// SIMATIC S7-200 project (STEP 7-Micro/WIN), CPU 221 REL 01.10

ORGANIZATION_BLOCK MAIN:OB1
TITLE=PROGRAM COMMENTS
BEGIN
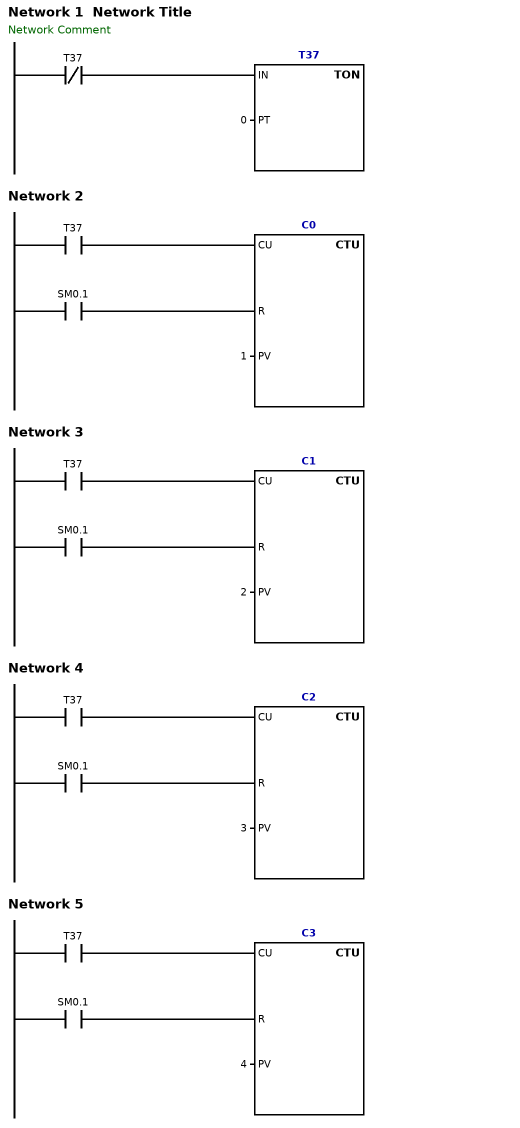
Network 1 // Network Title
// Network Comment
// (network saved uncompiled; LAD cells follow)
// row 0: c0 -|/|- T37  c1 --  c2 [TON T37 IN:=power@row0, PT:=0]
// row 1: c2 [box]
Network 2
LD     T37
LD     SM0.1
CTU    C0, 1
Network 3
LD     T37
LD     SM0.1
CTU    C1, 2
Network 4
LD     T37
LD     SM0.1
CTU    C2, 3
Network 5
LD     T37
LD     SM0.1
CTU    C3, 4
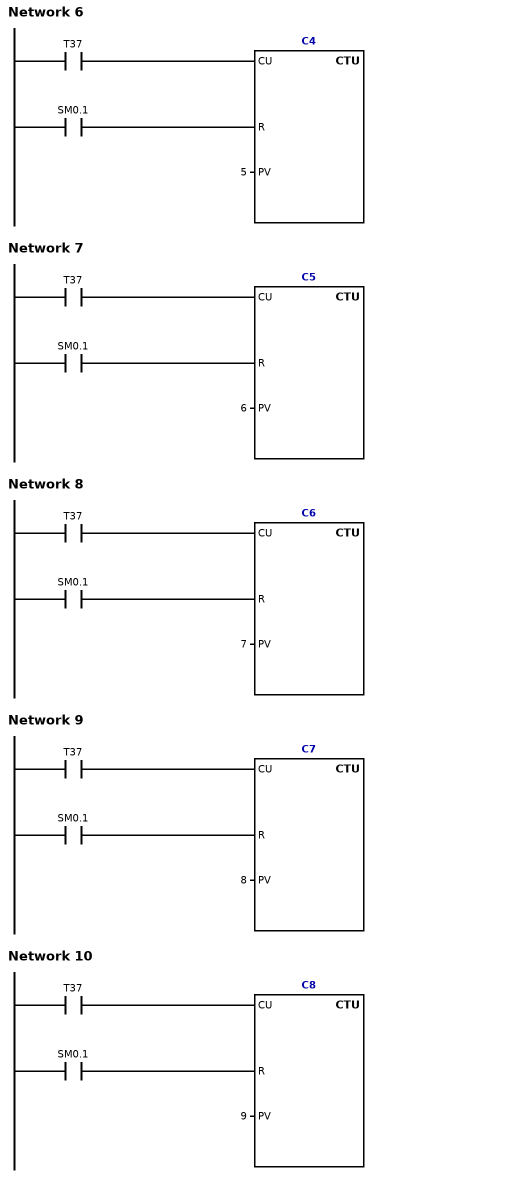
Network 6
LD     T37
LD     SM0.1
CTU    C4, 5
Network 7
LD     T37
LD     SM0.1
CTU    C5, 6
Network 8
LD     T37
LD     SM0.1
CTU    C6, 7
Network 9
LD     T37
LD     SM0.1
CTU    C7, 8
Network 10
LD     T37
LD     SM0.1
CTU    C8, 9
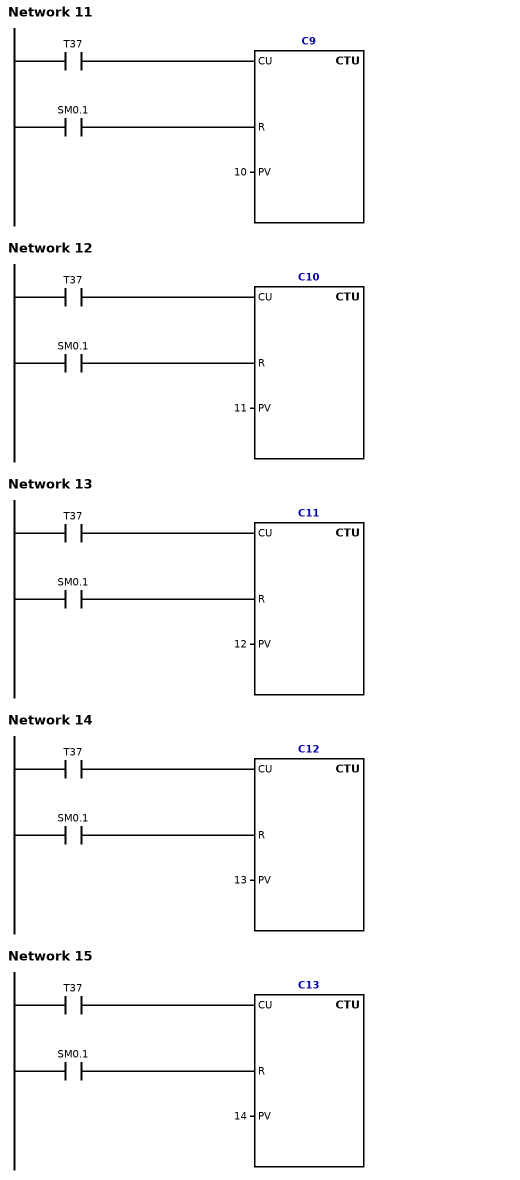
Network 11
LD     T37
LD     SM0.1
CTU    C9, 10
Network 12
LD     T37
LD     SM0.1
CTU    C10, 11
Network 13
LD     T37
LD     SM0.1
CTU    C11, 12
Network 14
LD     T37
LD     SM0.1
CTU    C12, 13
Network 15
LD     T37
LD     SM0.1
CTU    C13, 14
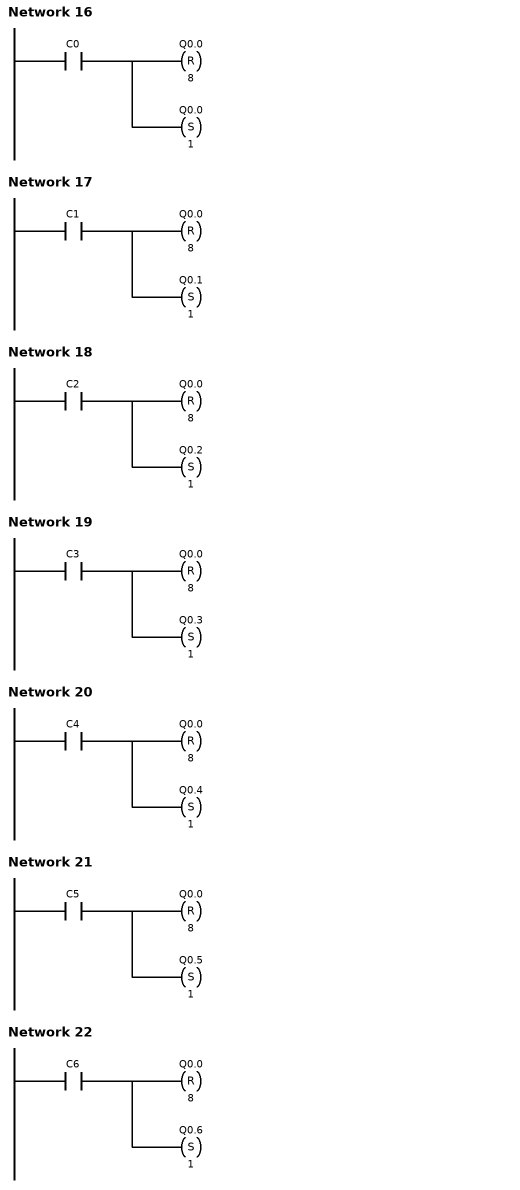
Network 16
LD     C0
R      Q0.0, 8
S      Q0.0, 1
Network 17
LD     C1
R      Q0.0, 8
S      Q0.1, 1
Network 18
LD     C2
R      Q0.0, 8
S      Q0.2, 1
Network 19
LD     C3
R      Q0.0, 8
S      Q0.3, 1
Network 20
LD     C4
R      Q0.0, 8
S      Q0.4, 1
Network 21
LD     C5
R      Q0.0, 8
S      Q0.5, 1
Network 22
LD     C6
R      Q0.0, 8
S      Q0.6, 1
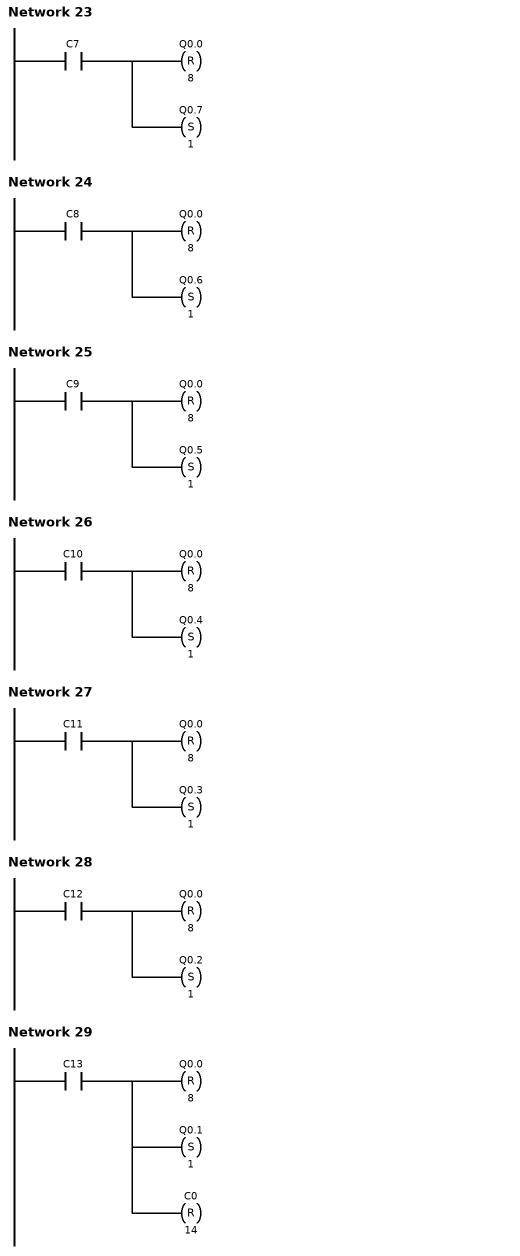
Network 23
LD     C7
R      Q0.0, 8
S      Q0.7, 1
Network 24
LD     C8
R      Q0.0, 8
S      Q0.6, 1
Network 25
LD     C9
R      Q0.0, 8
S      Q0.5, 1
Network 26
LD     C10
R      Q0.0, 8
S      Q0.4, 1
Network 27
LD     C11
R      Q0.0, 8
S      Q0.3, 1
Network 28
LD     C12
R      Q0.0, 8
S      Q0.2, 1
Network 29
LD     C13
R      Q0.0, 8
S      Q0.1, 1
R      C0, 14
END_ORGANIZATION_BLOCK
